FUNCTION_BLOCK TestFB// IMPLEMENTS ITestProps
VAR_INPUT
END_VAR
VAR_OUTPUT
END_VAR
VAR
END_VAR

END_FUNCTION_BLOCK

(* stored: Version 1.1.0.1, ProductVersion 3.1.4024.11
   POU TestFB: Id {d4512a1f-eebd-4ae3-84c4-0871c2262757}, SpecialFunc None *)
